PROGRAM LOAD_FUKUDA_1
VAR_INPUT

END_VAR

VAR
	TMR_DELAY: TON;
	TMR1:TON;
END_VAR

CASE INPUT_VAR.I_CASE OF
0: //standby near lotbox
	IF INPUT_VAR.ACTIVE_ID=6 THEN
		INPUT_VAR.ACTIVE_ID:=1;
	END_IF
	CASE INPUT_VAR.I_CURRENT_TRANSACTION.TRANSPORT_INDEX OF
		2 : FUKUDA_MOVE(STEP_DATA_1:=INPUT_VAR.I_CURRENT_TRANSACTION.STATION_NUMBER_LOAD,
				STEP_DATA_2:=3,
				STEP_DATA_3:=INPUT_VAR.I_CURRENT_TRANSACTION.JIG_INDEX_LOAD,
				STEP_DATA_4:=0,
				STEP_DATA_5:=1);
		1 : FUKUDA_MOVE(STEP_DATA_1:=INPUT_VAR.I_CURRENT_TRANSACTION.STATION_NUMBER_LOAD,
				STEP_DATA_2:=3,
				STEP_DATA_3:=INPUT_VAR.I_CURRENT_TRANSACTION.JIG_INDEX_LOAD,
				STEP_DATA_4:=1,
				STEP_DATA_5:=0);
				
	input_var.O_VACUUM_On:=FALSE;
	input_var.O_VACUUM_OFF:=FALSE;	
	TMR_DELAY(IN:=FALSE);

	END_CASE
				
1: //standby near lotbox
	
	IF INPUT_VAR.ACTIVE_ID=6 THEN
		INPUT_VAR.ACTIVE_ID:=1;
	END_IF
		FUKUDA_MOVE(STEP_DATA_1:=INPUT_VAR.I_CURRENT_TRANSACTION.STATION_NUMBER_LOAD,
				STEP_DATA_2:=4,
				STEP_DATA_3:=INPUT_VAR.I_CURRENT_TRANSACTION.JIG_INDEX_LOAD,
				STEP_DATA_4:=0,
				STEP_DATA_5:=0);

		CASE INPUT_VAR.I_CURRENT_TRANSACTION.TRANSPORT_INDEX OF
		1:
			INPUT_VAR.I_LOADING_DONE_A:=FALSE;
		
		2:
			INPUT_VAR.I_LOADING_DONE_B:=FALSE;
	END_CASE

		
				
2://vacuum position 
	IF INPUT_VAR.ACTIVE_ID=6 THEN
		INPUT_VAR.ACTIVE_ID:=1;
	END_IF
	FUKUDA_MOVE(STEP_DATA_1:=INPUT_VAR.I_CURRENT_TRANSACTION.STATION_NUMBER_LOAD,
				STEP_DATA_2:=4,
				STEP_DATA_3:=INPUT_VAR.I_CURRENT_TRANSACTION.JIG_INDEX_LOAD,
				STEP_DATA_4:=0,
				STEP_DATA_5:=0);
	IF INPUT_VAR.ACTIVE_ID=3 THEN
		input_var.O_VACUUM_ON:=TRUE;
		input_var.O_VACUUM_OFF:=FALSE;	
	END_IF

3://vacuum position 
	IF INPUT_VAR.ACTIVE_ID=6 THEN
		INPUT_VAR.ACTIVE_ID:=1; 
	END_IF
	FUKUDA_MOVE(STEP_DATA_1:=INPUT_VAR.I_CURRENT_TRANSACTION.STATION_NUMBER_LOAD,
				STEP_DATA_2:=4,
				STEP_DATA_3:=INPUT_VAR.I_CURRENT_TRANSACTION.JIG_INDEX_LOAD,
				STEP_DATA_4:=0,
				STEP_DATA_5:=0);
	
 		
//CHECK JIG FUKUDA PRESENCE			
	IF  input_var.O_VACUUM_ON THEN
		TMR1(IN:=TRUE,PT:=T#2S);
		IF TMR1.Q THEN
			IF NOT INPUT_VAR.I_VACUUM_ON AND input_var.O_VACUUM_ON THEN
				INPUT_VAR.JIG_FUKUDA_PRESENCE :=TRUE;
			ELSE
				INPUT_VAR.JIG_FUKUDA_PRESENCE :=FALSE;	
				FUKUDA_MOVE(STEP_DATA_1:=INPUT_VAR.I_CURRENT_TRANSACTION.STATION_NUMBER_LOAD,
				STEP_DATA_2:=2,
				STEP_DATA_3:=INPUT_VAR.I_CURRENT_TRANSACTION.JIG_INDEX_LOAD,
				STEP_DATA_4:=0,
				STEP_DATA_5:=0);
				
				FUKUDA_MOVE(STEP_DATA_1:=INPUT_VAR.I_CURRENT_TRANSACTION.STATION_NUMBER_LOAD,
				STEP_DATA_2:=1,
				STEP_DATA_3:=INPUT_VAR.I_CURRENT_TRANSACTION.JIG_INDEX_LOAD,
				STEP_DATA_4:=0,
				STEP_DATA_5:=0);
			input_var.O_VACUUM_ON:=FALSE;
			input_var.O_VACUUM_OFF:=FALSE;
			TMR_DELAY(IN:=TRUE,PT:=T#2.5S);
		
			IF TMR_DELAY.Q THEN
				FLAG_VAR.ALLOW_EXECUTE_LOAD_FUKUDA:=FALSE;
				INPUT_VAR.I_CURRENT_TRANSACTION.JIG_INDEX_LOAD:=INPUT_VAR.I_CURRENT_TRANSACTION.JIG_INDEX_LOAD+0;
				INPUT_VAR.I_CASE:=0;
			END_IF
		END_IF
	ELSE
		TMR1(IN:=FALSE);	
	END_IF 
		
				//INPUT_VAR.JIG_FUKUDA_PRESENCE :=TRUE;
				//IF INPUT_VAR.I_CURRENT_TRANSACTION.JIG_INDEX_LOAD >=11 THEN
					//INPUT_VAR.I_CASE:=100;
			
				//FLAG_VAR.ALLOW_EXECUTE_LOAD_FUKUDA:=FALSE;
				//INPUT_VAR.I_CASE:=0;
				//INPUT_VAR.I_CURRENT_TRANSACTION.JIG_INDEX_LOAD:=1 ;
					//ELSE
						
				//END_IF
				
				//TMR_DELAY(IN:=FALSE);
				//LOAD_FUKUDA();
				//FLAG_VAR.ALLOW_EXECUTE_LOAD_FUKUDA:=FALSE;
	
	END_IF
 
	
4://vacuum position 
	IF INPUT_VAR.ACTIVE_ID=6 THEN
		INPUT_VAR.ACTIVE_ID:=1;
	END_IF
	
	FUKUDA_MOVE(STEP_DATA_1:=7,
				STEP_DATA_2:=4,
				STEP_DATA_3:=INPUT_VAR.I_CURRENT_TRANSACTION.JIG_INDEX_LOAD,
				STEP_DATA_4:=0,
				STEP_DATA_5:=0);
				

5://vacuum position 
	IF INPUT_VAR.ACTIVE_ID=6 THEN
		INPUT_VAR.ACTIVE_ID:=1;
	END_IF
	
	FUKUDA_MOVE(STEP_DATA_1:=8,
				STEP_DATA_2:=2,
				STEP_DATA_3:=INPUT_VAR.I_CURRENT_TRANSACTION.JIG_INDEX_LOAD,
				STEP_DATA_4:=0,
				STEP_DATA_5:=0);
	
6://gripping position
	IF INPUT_VAR.ACTIVE_ID=6 THEN
		INPUT_VAR.ACTIVE_ID:=1;
	END_IF

	FUKUDA_MOVE(STEP_DATA_1:=INPUT_VAR.I_CURRENT_TRANSACTION.TRANSPORT_INDEX+4,
				STEP_DATA_2:=2,
				STEP_DATA_3:=12,
				STEP_DATA_4:=0,
				STEP_DATA_5:=0);


7://placing onto fukuda transport
	IF INPUT_VAR.ACTIVE_ID=6 THEN
		INPUT_VAR.ACTIVE_ID:=1;
	END_IF
	FUKUDA_MOVE(STEP_DATA_1:=INPUT_VAR.I_CURRENT_TRANSACTION.TRANSPORT_INDEX+4,
				STEP_DATA_2:=2,
				STEP_DATA_3:=11,
				STEP_DATA_4:=0,
				STEP_DATA_5:=0);

8://placing onto fukuda transport
	IF INPUT_VAR.ACTIVE_ID=6 THEN
		INPUT_VAR.ACTIVE_ID:=1;
	END_IF
	
	FUKUDA_MOVE(STEP_DATA_1:=INPUT_VAR.I_CURRENT_TRANSACTION.TRANSPORT_INDEX+4,
				STEP_DATA_2:=2,
				STEP_DATA_3:=11,
				STEP_DATA_4:=0,
				STEP_DATA_5:=0);
	IF INPUT_VAR.ACTIVE_ID=3 THEN
		input_var.O_VACUUM_On:=FALSE;
		input_var.O_VACUUM_OFF:=TRUE;	
	END_IF

	
9://homing
	IF INPUT_VAR.ACTIVE_ID=6 THEN
		INPUT_VAR.ACTIVE_ID:=1;
	END_IF
	
	FUKUDA_MOVE(STEP_DATA_1:=INPUT_VAR.I_CURRENT_TRANSACTION.TRANSPORT_INDEX+4,
				STEP_DATA_2:=1,
				STEP_DATA_3:=11,
				STEP_DATA_4:=0,
				STEP_DATA_5:=0);
			
				
10://pusH fukuda transport
	IF INPUT_VAR.ACTIVE_ID=6 THEN
		INPUT_VAR.ACTIVE_ID:=1;
	END_IF
	input_var.O_VACUUM_OFF:=FALSE;
	CASE INPUT_VAR.I_CURRENT_TRANSACTION.TRANSPORT_INDEX OF
		2 : FUKUDA_MOVE(STEP_DATA_1:=0,
				STEP_DATA_2:=0,
				STEP_DATA_3:=0,
				STEP_DATA_4:=0,
				STEP_DATA_5:=2);
		1 : FUKUDA_MOVE(STEP_DATA_1:=0,
				STEP_DATA_2:=0,
				STEP_DATA_3:=0,
				STEP_DATA_4:=2,
				STEP_DATA_5:=0);
	END_CASE			 

100:

	input_var.O_VACUUM_On:=FALSE;
	input_var.O_VACUUM_OFF:=FALSE;	
	
END_CASE 
IF INPUT_VAR.I_CASE=11 THEN
			CASE INPUT_VAR.I_CURRENT_TRANSACTION.TRANSPORT_INDEX OF
		1:	
			IF INPUT_VAR.I_FUKUDA_TRANSFER_AT_FRONT_A THEN
				INPUT_VAR.I_LOADING_DONE_A:=TRUE;
				IF  INPUT_VAR.I_LOADING_DONE_A THEN
					FLAG_VAR.ALLOW_EXECUTE_LOAD_FUKUDA:=FALSE;			
					INPUT_VAR.I_CASE:=100;
				END_IF
			END_IF
			
				2:
			IF INPUT_VAR.I_FUKUDA_TRANSFER_AT_FRONT_B THEN
				INPUT_VAR.I_LOADING_DONE_B:=TRUE;
				IF  INPUT_VAR.I_LOADING_DONE_B THEN
					FLAG_VAR.ALLOW_EXECUTE_LOAD_FUKUDA:=FALSE;			
					INPUT_VAR.I_CASE:=100;
				END_IF
			END_IF
			
	END_CASE

END_IF

END_PROGRAM

(* stored: Version 1.1.0.1, ProductVersion 3.1.4020.12
   POU LOAD_FUKUDA_1: Id {5a50fe34-120f-4a70-a4ac-83f1b925638f}, SpecialFunc None *)
